FUNCTION Convert_UDINT_TO_DT : Hresult
VAR_INPUT
	in : UDINT;
	out : REFERENCE TO DT;
END_VAR
VAR
	converted : DT;
END_VAR

converted := UDINT_TO_DT(in);

IF (DT_TO_UDINT(converted) <> in) THEN
	Convert_UDINT_TO_DT := INCOMPATIBLE;
	RETURN;
END_IF

out := converted;

END_FUNCTION

(* stored: Version 1.1.0.1, ProductVersion 3.1.4024.12
   POU Convert_UDINT_TO_DT: Id {8d1103fb-ff82-4179-af44-2af0cd2fd0c0}, SpecialFunc None *)
